// TwinCAT 3 PLC project PLC
// ProgramVersion: 3.1.4026.20
// CompilerDefines: VISU_USEPROPERTYINFO
// libraries:
//   Tc2_Standard, * (Beckhoff Automation GmbH)
//   Tc2_System, * (Beckhoff Automation GmbH)
//   Tc3_Vision, * (Beckhoff Automation GmbH)
//   VisuSymbols, 4.5.0.0 (System)
// project tree:
//   / GlobalTextList.TcGTLO, MAIN.TcPOU, PlcTask.TcTTO, Visualization Manager.TcVMO (not stored)
//   GVLs/ GVL.TcGVL
//   Source/debug/ CheckBounds.TcPOU (not stored)
//   Source/EL2574/DUT/ ST_EL2574_ExtendedMode.TcDUT, ST_EL2574_In.TcDUT, ST_EL2574_Out.TcDUT
//   Source/EL2574/ EL2574_ExtendedMode.TcPOU, I_EL2574_CommandMode.TcIO
//   Source/ImageSerializer/Base/ ImageSerializer.TcPOU
//   Source/ImageSerializer/Interfaces/ I_ImageSerializer.TcIO
//   Source/ImageSerializer/Matrix/ MatrixImageSerializer.TcPOU
//   Source/ImageSerializer/Null/ NullImageSerializer.TcPOU
//   Source/Library/Animation/ I_Animation.TcIO, SpriteSheetAnimationFrames.TcPOU
//   Source/Library/BlendModes/ BaseBlender.TcPOU, I_ImageBlender.TcIO, LerpMixer.TcPOU, MultiplyMixer.TcPOU
//   Source/Library/ Modulate.TcPOU
//   Source/Library/Scene/ Scene.TcPOU
//   Source/PixelReader/ EL2574PixelReader.TcPOU, I_PixelReader.TcIO
//   Source/ ST_Colors.TcDUT, U_Pixel.TcDUT
//   Source/Unwrappers/ I_Unwrapper.TcIO, RepeatUnwrap.TcPOU, ExtendUnwrap.TcPOU, ReflectUnwrap.TcPOU
//   VISUs/ UC_Slider.TcVIS, Visualization.TcVIS
// real-time tasks:
//   TASK PlcTask: cycle T#1ms, priority 20, ADS port 350
// I/O:
//   DEVICE Device 2 (EtherCAT), AmsNetId 192.168.1.242.3.1
//     Term 1 (EK1200) [EK1200-5000 EtherCAT Power supply (2A E-Bus)]
//       Term 3 (EL2574) [EL2574 4 Ch. Pixel LED Controller]
//         modules: SlotGroup 1 (Slot 1, 2) (1xASYNC), SlotGroup 1 (Slot 1, 2) (1xASYNC), SlotGroup 2 (Slot 3, 4) (EMPTY2), SlotGroup 2 (Slot 3, 4) (EMPTY2)
//       Term 3 (EL9011) [EL9011 End Terminal]
// variable links:
//   (this object) <-> Device 2 (EtherCAT)/Term 1 (EK1200)/Term 3 (EL2574)
//     PlcTask Inputs/MAIN.el2574_ch1.pdo.In/Busy <-> SlotGroup 1 (Slot 1, 2) (1xASYNC)/Status Channel 1/Status/Busy
//     PlcTask Inputs/MAIN.el2574_ch1.pdo.In/CommandAck <-> SlotGroup 1 (Slot 1, 2) (1xASYNC)/Status Channel 1/Status/Command Acknowledge
//     PlcTask Inputs/MAIN.el2574_ch1.pdo.In/CommandReject <-> SlotGroup 1 (Slot 1, 2) (1xASYNC)/Status Channel 1/Status/Command Reject
//     PlcTask Inputs/MAIN.el2574_ch1.pdo.In/Error <-> SlotGroup 1 (Slot 1, 2) (1xASYNC)/Status Channel 1/Status/Error
//     PlcTask Inputs/MAIN.el2574_ch1.pdo.In/InputCycleCounter <-> SlotGroup 1 (Slot 1, 2) (1xASYNC)/Status Channel 1/Status/Input Cycle Counter
//     PlcTask Inputs/MAIN.el2574_ch1.pdo.In/SendAck <-> SlotGroup 1 (Slot 1, 2) (1xASYNC)/Status Channel 1/Status/Send Acknowledge
//     PlcTask Inputs/MAIN.el2574_ch1.pdo.In/Transmit <-> SlotGroup 1 (Slot 1, 2) (1xASYNC)/Status Channel 1/Status/Transmit
//     PlcTask Inputs/MAIN.el2574_ch1.pdo.In/UpdateAck <-> SlotGroup 1 (Slot 1, 2) (1xASYNC)/Status Channel 1/Status/Update Acknowledge
//     PlcTask Inputs/MAIN.el2574_ch1.pdo.In/Warning <-> SlotGroup 1 (Slot 1, 2) (1xASYNC)/Status Channel 1/Status/Warning
//     PlcTask Outputs/MAIN.el2574_ch1.pdo.Out/Execute <-> SlotGroup 1 (Slot 1, 2) (1xASYNC)/Extended Channel 1/Extended Control/Execute
//     PlcTask Outputs/MAIN.el2574_ch1.pdo.Out/Index <-> SlotGroup 1 (Slot 1, 2) (1xASYNC)/Extended Channel 1/Extended Control/Index
//     PlcTask Outputs/MAIN.el2574_ch1.pdo.Out/Segment <-> SlotGroup 1 (Slot 1, 2) (1xASYNC)/Extended Channel 1/Extended Control/Segment
//     PlcTask Outputs/MAIN.el2574_ch1.pdo.Out/Send <-> SlotGroup 1 (Slot 1, 2) (1xASYNC)/Extended Channel 1/Extended Control/Send
//     PlcTask Outputs/MAIN.el2574_ch1.pdo.Out/Update <-> SlotGroup 1 (Slot 1, 2) (1xASYNC)/Extended Channel 1/Extended Control/Update
//     PlcTask Outputs/MAIN.el2574_ch1.pdo.Out/Write <-> SlotGroup 1 (Slot 1, 2) (1xASYNC)/Extended Channel 1/Extended Control/Write

CONFIGURATION PLC
    RESOURCE PLC ON TwinCAT3
        TASK PlcTask(INTERVAL := T#1ms, PRIORITY := 20);
        PROGRAM MAIN WITH PlcTask : MAIN;
    END_RESOURCE
END_CONFIGURATION

// ---- Source/EL2574/DUT/ST_EL2574_ExtendedMode.TcDUT
TYPE ST_EL2574_ExtendedMode :
	STRUCT
		In	AT %I* : ST_EL2574_In;
		Out AT %Q* : ST_EL2574_Out;
	END_STRUCT
END_TYPE

// ---- Source/EL2574/DUT/ST_EL2574_In.TcDUT
TYPE ST_EL2574_In :
	STRUCT
		Busy			  : BIT;
		Transmit		  : BIT;
		SendAck			  : BIT;
		UpdateAck		  : BIT;
		CommandAck		  : BIT;
		CommandReject	  : BIT;
		Warning			  : BIT;
		Error			  : BIT;
		InputCycleCounter : BYTE;
	END_STRUCT
END_TYPE

// ---- Source/EL2574/DUT/ST_EL2574_Out.TcDUT
TYPE ST_EL2574_Out :
	STRUCT
		Execute : BIT;
		Send	: BIT;
		Update	: BIT;
		Write	: BIT;
		Index	: USINT;
		Segment : ARRAY[0..7] OF UDINT;
	END_STRUCT
END_TYPE

// ---- Source/ST_Colors.TcDUT
TYPE ST_Colors :
	STRUCT
		Red	  : BYTE;
		Green : BYTE;
		Blue  : BYTE;
		White : BYTE;
	END_STRUCT
END_TYPE

// ---- Source/U_Pixel.TcDUT
TYPE U_Pixel : UNION
		Pdo	   : UDINT;
		Colors : ST_Colors;
	END_UNION
END_TYPE

// ---- GVLs/GVL.TcGVL
VAR_GLOBAL CONSTANT
	STRIP_LENGTH : UDINT := 12;
END_VAR

// ---- Source/EL2574/I_EL2574_CommandMode.TcIO
INTERFACE I_EL2574_CommandMode

METHOD PUBLIC ClearAll : I_EL2574_CommandMode
VAR_INPUT
END_VAR
END_METHOD

METHOD PUBLIC ColorGradient2Point : I_EL2574_CommandMode
VAR_INPUT
	StartPosition : UINT;
	NumberOfPixels : UINT;
	Color1 : STRING(9);
	Color2 : STRING(9);
END_VAR
END_METHOD

METHOD PUBLIC ColorGradient3Point : I_EL2574_CommandMode
VAR_INPUT
	StartPosition : UINT;
	NumberOfPixels : UINT;
	Color1 : STRING(9);
	Color2 : STRING(9);
	Color3 : STRING(9);
END_VAR
END_METHOD

METHOD PUBLIC ColorGradient4Point : I_EL2574_CommandMode
VAR_INPUT
	StartPosition : UINT;
	NumberOfPixels : UINT;
	Color1 : STRING(9);
	Color2 : STRING(9);
	Color3 : STRING(9);
	Color4 : STRING(9);
END_VAR
END_METHOD

METHOD PUBLIC CopyPixels : I_EL2574_CommandMode
VAR_INPUT
	StartPosition : UINT;
	NumberOfPixels : UINT;
	TargetPosition : UINT;
END_VAR
END_METHOD

METHOD PUBLIC FillColor : I_EL2574_CommandMode
VAR_INPUT
	StartPosition : UINT;
	NumberOfPixels : UINT;
	Red : USINT;
	Green : USINT;
	Blue : USINT;
	White : USINT;
END_VAR
END_METHOD

METHOD PUBLIC Invert : I_EL2574_CommandMode
VAR_INPUT
	StartPosition : UINT;
	NumberOfPixels : UINT;
END_VAR
END_METHOD

METHOD PUBLIC MovePixels : I_EL2574_CommandMode
VAR_INPUT
	StartPosition : UINT;
	NumberOfPixels : UINT;
	TargetPosition : UINT;
END_VAR
END_METHOD

METHOD PUBLIC RotateLeft : I_EL2574_CommandMode
VAR_INPUT
	StartPosition : UINT;
	NumberOfPixels : UINT;
	Shift : UINT;
END_VAR
END_METHOD

METHOD PUBLIC RotateRight : I_EL2574_CommandMode
VAR_INPUT
	StartPosition : UINT;
	NumberOfPixels : UINT;
	Shift : UINT;
END_VAR
END_METHOD

METHOD PUBLIC Send : I_EL2574_CommandMode
VAR_INPUT
END_VAR
END_METHOD

METHOD PUBLIC SendAndUpdate : I_EL2574_CommandMode
VAR_INPUT
END_VAR
END_METHOD

METHOD PUBLIC Update : I_EL2574_CommandMode
VAR_INPUT
END_VAR
END_METHOD

END_INTERFACE

// ---- Source/ImageSerializer/Interfaces/I_ImageSerializer.TcIO
INTERFACE I_ImageSerializer

METHOD PUBLIC ConnectTo
VAR_INPUT
	ImageSerializer : I_ImageSerializer;
END_VAR
END_METHOD

METHOD PUBLIC GetTotalSerializablePixelCount : UDINT
VAR_INPUT
END_VAR
END_METHOD

PROPERTY PUBLIC PixelCount : UDINT
GET
END_GET
END_PROPERTY

METHOD PUBLIC TryGetPixel : BOOL
VAR_INPUT
	PixelIndex : UDINT;
	Reader : I_PixelReader;
END_VAR
END_METHOD

METHOD PUBLIC UpdateImage
VAR_INPUT
	Source : ITcVnImage;
END_VAR
END_METHOD

END_INTERFACE

// ---- Source/Library/Animation/I_Animation.TcIO
INTERFACE I_Animation

PROPERTY PUBLIC CurrentFrameImage : ITcVnImage
GET
END_GET
END_PROPERTY

PROPERTY PUBLIC CurrentFrameIndex : UDINT
GET
END_GET
END_PROPERTY

PROPERTY PUBLIC IsAtLastFrame : BOOL
GET
END_GET
END_PROPERTY

METHOD PUBLIC MoveToStart
VAR_INPUT
END_VAR
END_METHOD

PROPERTY PUBLIC TotalFrameCount : UDINT
GET
END_GET
END_PROPERTY

METHOD PUBLIC TryMoveNext : BOOL
VAR_INPUT
END_VAR
END_METHOD

METHOD PUBLIC TryMovePrevious : BOOL
VAR_INPUT
END_VAR
END_METHOD

END_INTERFACE

// ---- Source/Library/BlendModes/I_ImageBlender.TcIO
INTERFACE I_ImageBlender

METHOD Mix
VAR_INPUT
	ImageBottomLayer : ITcVnImage;
	ImageTopLayer	 : ITcVnImage;
END_VAR
END_METHOD

END_INTERFACE

// ---- Source/PixelReader/I_PixelReader.TcIO
INTERFACE I_PixelReader

PROPERTY PUBLIC Value : Reference to TcVnVector4_LREAL
GET
END_GET
END_PROPERTY

END_INTERFACE

// ---- Source/Unwrappers/I_Unwrapper.TcIO
INTERFACE I_Unwrapper

METHOD Sample : BOOL
VAR_INPUT
	ImageWidth, ImageHeight	  : UDINT;
	XOffset, YOffset		  : UDINT;
END_VAR
END_METHOD

PROPERTY X : UDINT
GET
END_GET
END_PROPERTY

PROPERTY Y : UDINT
GET
END_GET
END_PROPERTY

END_INTERFACE

// ---- MAIN.TcPOU
PROGRAM MAIN
VAR
	// --- Sprite source images ---
	Black	   : SpriteSheetAnimationFrames(SpriteSheetFilePath := 'C:\temp\images\black_64x1.png', SpriteWidth := 64, SpriteHeight := 1, TotalSprites := 1, Columns := 1, Rows := 1);
	Red		   : SpriteSheetAnimationFrames(SpriteSheetFilePath := 'C:\temp\images\red_64x1.png', SpriteWidth := 64, SpriteHeight := 1, TotalSprites := 1, Columns := 1, Rows := 1);
	Blue	   : SpriteSheetAnimationFrames(SpriteSheetFilePath := 'C:\temp\images\blue_64x1.png', SpriteWidth := 64, SpriteHeight := 1, TotalSprites := 1, Columns := 1, Rows := 1);
	Green	   : SpriteSheetAnimationFrames(SpriteSheetFilePath := 'C:\temp\images\green_64x1.png', SpriteWidth := 64, SpriteHeight := 1, TotalSprites := 1, Columns := 1, Rows := 1);
	Background : SpriteSheetAnimationFrames(SpriteSheetFilePath := 'C:\temp\images\rainbow_gradient.png', SpriteWidth := 1000, SpriteHeight := 1, TotalSprites := 1, Columns := 1, Rows := 1);
	white	   : SpriteSheetAnimationFrames(SpriteSheetFilePath := 'C:\temp\images\whitealpha3_32_32.png', SpriteWidth := 32, SpriteHeight := 1, TotalSprites := 1, Columns := 1, Rows := 1);
	shortred   : SpriteSheetAnimationFrames(SpriteSheetFilePath := 'C:\temp\images\shortred_32_32.png', SpriteWidth := 32, SpriteHeight := 1, TotalSprites := 1, Columns := 1, Rows := 1);

	// --- Modulators (scroll/unwrap each source into a strip-length output) ---
	ModulateBackground : Modulate(Width := GVL.STRIP_LENGTH);
	ShortredModulator  : Modulate(Width := GVL.STRIP_LENGTH);
	WhiteModulator	   : Modulate(Width := GVL.STRIP_LENGTH);
	backgroundOffset   : UDINT;
	shortredOffset	   : UDINT;
	shortedRollOver	   : UDINT;
	whiteOffset		   : UDINT;
	whiteRollOver	   : UDINT;
	redOffset		   : UDINT;
	blueOffset		   : UDINT;
	greenOffset		   : UDINT;
	UpdateBackground   : BOOL;
	UpdateShortred	   : BOOL;
	UpdateWhite		   : BOOL;
	UpdateRed		   : BOOL;
	UpdateBlue		   : BOOL;
	UpdateGreen		   : BOOL;

	// --- Scene compositor ---
	MyScene : Scene;
	lerp	: LerpMixer;
	weight	: LREAL := 0.85;

	// --- Displayable image handles (for scope/HMI monitoring) ---
	SceneImage		  : ITcVnDisplayableImage;
	displayBackground : ITcVnDisplayableImage;
	displayShortred	  : ITcVnDisplayableImage;
	displayWhite	  : ITcVnDisplayableImage;
	displayRed		  : ITcVnDisplayableImage;
	displayBlue		  : ITcVnDisplayableImage;
	displayGreen	  : ITcVnDisplayableImage;

	// --- Animation timing ---
	Animate			 : BOOL := TRUE;
	AddBlackLayer	 : BOOL := FALSE;
	AnimateBackgroud : BOOL := TRUE;
	AddBackground	 : BOOL := TRUE;
	BackgroundRate	 : TON	:= (PT := T#80MS);
	AddShortedLayer	 : BOOL := TRUE;
	ShortredRate	 : TON	:= (PT := T#200MS);
	AddWhiteLayer	 : BOOL := TRUE;
	WhiteRate		 : TON	:= (PT := T#150MS);
	AddRedLayer		 : BOOL := FALSE;
	AddBlueLayer	 : BOOL := FALSE;
	AddGreenLayer	 : BOOL := FALSE;

	// --- Unwrap modes ---
	unwraptype			: UDINT;
	reflect				: ReflectUnwrap;
	RepeatNormal		: RepeatUnwrap;
	Extend				: ExtendUnwrap;
	width, height, x, y : UDINT; // reflect.Sample inputs

	// --- Hardware ---
	LEDStrip   : MatrixImageSerializer(Height := 1, Width := GVL.STRIP_LENGTH, X := 0, Y := 0, FlipX := FALSE, FlipY := FALSE, Rotate := FALSE);
	el2574_ch1 : EL2574_ExtendedMode(TotalPixels := GVL.STRIP_LENGTH);

	// --- Misc ---
	val	   : HRESULT;
	format : TcVnPixelFormat;
END_VAR

_AppInfo.KeepOutputsOnBP := TRUE;
// 1. LOAD GUARD — wait until all sprite sheets are ready
IF NOT Black.TryLoad() OR NOT Background.TryLoad() OR NOT shortred.TryLoad() OR NOT white.TryLoad() OR NOT Red.TryLoad() OR NOT Blue.TryLoad() OR NOT Green.TryLoad() THEN
	RETURN;
END_IF

// 2. ANIMATION TICK — advance offsets at each layer's own rate
ShortredRate(IN := NOT ShortredRate.Q AND Animate);
IF ShortredRate.Q THEN
	shortredOffset := shortredOffset + 1;
	IF shortredOffset >= shortedRollOver THEN
		shortredOffset := 0;
	END_IF

	UpdateShortred := TRUE;
END_IF

WhiteRate(IN := NOT WhiteRate.Q AND Animate);
IF WhiteRate.Q THEN
	whiteOffset := whiteOffset + 1;
	IF whiteOffset >= whiteRollOver THEN
		whiteOffset := 0;
	END_IF

	UpdateWhite := TRUE;
END_IF

BackgroundRate(IN := NOT BackgroundRate.Q AND Animate AND AnimateBackgroud);
IF BackgroundRate.Q THEN
	backgroundOffset := backgroundOffset + 1;
	UpdateBackground := TRUE;
END_IF

// 3. UNWRAP MODE SELECT — override shortred/white unwrapper at runtime
ModulateBackground.Unwrapper := reflect;
CASE unwraptype OF
	0:
		shortedRollOver				:= 32;
		whiteRollOver				:= 32;
		ShortredModulator.Unwrapper := RepeatNormal;
		WhiteModulator.Unwrapper	:= RepeatNormal;

	1:
		shortedRollOver				:= GVL.STRIP_LENGTH;
		whiteRollOver				:= GVL.STRIP_LENGTH;
		ShortredModulator.Unwrapper := reflect;
		WhiteModulator.Unwrapper	:= reflect;

	2:
		ShortredModulator.Unwrapper := Extend;
		WhiteModulator.Unwrapper	:= Extend;

END_CASE

// 4. MODULATE — scroll each source into a strip-length output frame
IF UpdateBackground OR NOT AnimateBackgroud THEN
	ModulateBackground.GetImage(Source		 := Background.CurrentFrameImage,
								SourceWidth	 := 1000,
								SourceHeight := 1,
								OutputWidth	 := GVL.STRIP_LENGTH,
								OutputHeight := 1,
								OffsetX		 := backgroundOffset,
								OffsetY		 := 0);

	UpdateBackground := FALSE;
END_IF

IF UpdateShortred THEN
	ShortredModulator.GetImage(shortred.CurrentFrameImage,
							   32,
							   1,
							   GVL.STRIP_LENGTH,
							   1,
							   shortredOffset,
							   0);

	UpdateShortred := FALSE;
END_IF

IF UpdateWhite THEN
	WhiteModulator.GetImage(white.CurrentFrameImage,
							32,
							1,
							GVL.STRIP_LENGTH,
							1,
							whiteOffset,
							0);

	UpdateWhite := FALSE;
END_IF

// 5. COMPOSE SCENE — stack layers onto background with lerp blend
IF NOT el2574_ch1.IsBusy THEN
	IF AddBlackLayer THEN
		MyScene.Initalize(Black.CurrentFrameImage);
	END_IF

	IF AddBackground THEN
		MyScene.Initalize(ModulateBackground.CurrentFrameImage);
	END_IF

	lerp.Weight := weight;
	
	IF AddWhiteLayer THEN
		MyScene.AddLayer(WhiteModulator.CurrentFrameImage, lerp);
	END_IF
	
	IF AddShortedLayer THEN
		MyScene.AddLayer(ShortredModulator.CurrentFrameImage, lerp);
	END_IF

	IF AddRedLayer THEN
		MyScene.AddLayer(Red.CurrentFrameImage, lerp);
	END_IF

	IF AddBlueLayer THEN
		MyScene.AddLayer(Blue.CurrentFrameImage, lerp);
	END_IF

	IF AddGreenLayer THEN
		MyScene.AddLayer(Green.CurrentFrameImage, lerp);
	END_IF

	LEDStrip.UpdateImage(MyScene.Image);
	el2574_ch1.TrySendPixelsFromSerializer(LEDStrip);

	// 6. COPY TO DISPLAY — push images to HMI/scope handles
	val := F_VN_CopyIntoDisplayableImage(MyScene.Image, SceneImage, s_ok);
	val := F_VN_CopyIntoDisplayableImage(ModulateBackground.CurrentFrameImage, displayBackground, s_ok);
	val := F_VN_CopyIntoDisplayableImage(ShortredModulator.CurrentFrameImage, displayShortred, s_ok);
	val := F_VN_CopyIntoDisplayableImage(WhiteModulator.CurrentFrameImage, displayWhite, s_ok);
END_IF

el2574_ch1.CyclicCall();

END_PROGRAM

// ---- Source/Library/Animation/SpriteSheetAnimationFrames.TcPOU
FUNCTION_BLOCK SpriteSheetAnimationFrames IMPLEMENTS I_Animation
VAR
	spriteSheetFilePath : T_MAXSTRING;
	spriteWidth			: UDINT;
	spriteHeight		: UDINT;
	totalSprites		: UDINT;
	columns				: UDINT;
	rows				: UDINT;
	spriteSheetImage	: ITcVnImage;
	readImage			: FB_VN_ReadImage;

	// animation variables
	_currentFrameIndex	 : UDINT;
	_currentFrameImage	 : ITcVnImage;
	_LoadedImageFromDisk : ITcVnDisplayableImage;
END_VAR

PROPERTY PUBLIC CurrentFrameImage : ITcVnImage
GET
CurrentFrameImage := _currentFrameImage;
END_GET
END_PROPERTY

PROPERTY PUBLIC CurrentFrameIndex : UDINT
GET
CurrentFrameIndex := _currentFrameIndex;
END_GET
END_PROPERTY

METHOD FB_init : BOOL
VAR_INPUT
	bInitRetains		: BOOL; // if TRUE, the retain variables are initialized (warm start / cold start)
	bInCopyCode			: BOOL; // if TRUE, the instance afterwards gets moved into the copy code (online change)
	SpriteSheetFilePath : T_MAXSTRING;
	SpriteWidth			: UDINT;
	SpriteHeight		: UDINT;
	TotalSprites		: UDINT;
	Columns				: UDINT;
	Rows				: UDINT;
END_VAR
THIS^.spriteSheetFilePath := SpriteSheetFilePath;
THIS^.spriteWidth		  := SpriteWidth;
THIS^.spriteHeight		  := SpriteHeight;
THIS^.totalSprites		  := TotalSprites;
THIS^.columns			  := Columns;
THIS^.rows				  := Rows;
END_METHOD

PROPERTY PUBLIC IsAtLastFrame : BOOL
GET
IF TotalFrameCount = 0 THEN
	IsAtLastFrame := TRUE;
	RETURN;
END_IF

IsAtLastFrame := CurrentFrameIndex = TotalFrameCount - 1;
END_GET
END_PROPERTY

METHOD PUBLIC MoveToStart
VAR_INPUT
END_VAR
_currentFrameIndex := 0;
TryGetSprite(_currentFrameIndex, _currentFrameImage);
END_METHOD

PROPERTY PUBLIC TotalFrameCount : UDINT
GET
TotalFrameCount := totalSprites;
END_GET
END_PROPERTY

METHOD PRIVATE TryGetSprite : BOOL
VAR_INPUT
	Index : UDINT;
	Destination : REFERENCE TO ITcVnImage;
END_VAR
VAR
	spriteX : UDINT;
	spriteY : UDINT;
	spriteColumn : UDINT;
	spriteRow : UDINT;
	result : HRESULT;
END_VAR
IF Index > TotalFrameCount - 1 THEN
	RETURN;
END_IF

spriteColumn := Index MOD columns;
spriteRow := Index / columns;

spriteX := spriteColumn * spriteWidth;
spriteY := spriteRow * spriteHeight;

result := F_VN_CopyImage(spriteSheetImage, _currentFrameImage, s_OK);
result := F_VN_SetRoi(spriteX, spriteY, spriteWidth, spriteHeight, _currentFrameImage, result);

TryGetSprite := Succeeded(result);
END_METHOD

METHOD PUBLIC TryLoad : BOOL
VAR
	i : UDINT;
END_VAR
// if we already have an image loaded, then we can early jump out as we know everything is done. 
IF spriteSheetImage <> 0 THEN
	TryLoad := TRUE;
	RETURN;
END_IF

IF spriteSheetFilePath = '' OR  spriteWidth = 0 OR spriteHeight = 0 OR totalSprites = 0 OR columns = 0 OR rows = 0 THEN
	// this is our sanity check, we return out if anything is bad.
	// if we pass this point we know we can use the variables confidently.
	RETURN;
END_IF

// we keep polling the read until an image is read.  If it faults due to error then we just sit here and never return true.
readImage(sFilePath := spriteSheetFilePath, ipDestImage := spriteSheetImage, bRead := TRUE, nTimeout := T#500MS);
IF readImage.bBusy THEN 
	RETURN;
END_IF

IF readImage.bError THEN 
	RETURN;
END_IF 

// at this point we should have an image, so we will do one final check before moving on.  
IF spriteSheetImage = 0 THEN
	RETURN;
END_IF

F_VN_CopyIntoDisplayableImage(ipSrcImage:=spriteSheetImage,ipDestImage:=_LoadedImageFromDisk,hrPrev:=S_OK);

// we have made it this far, which means we need to set the CurrentFrameImage to the first part of the image and report as done. 
MoveToStart();
TryLoad := TRUE;
END_METHOD

METHOD PUBLIC TryMoveNext : BOOL
VAR_INPUT
END_VAR
IF _currentFrameIndex = TotalFrameCount - 1 THEN
	RETURN;
END_IF

_currentFrameIndex := _currentFrameIndex + 1;
TryMoveNext := TryGetSprite(_currentFrameIndex, _currentFrameImage);
END_METHOD

METHOD PUBLIC TryMovePrevious : BOOL
VAR_INPUT
END_VAR
IF _currentFrameIndex = 0 THEN
	RETURN;
END_IF

_currentFrameIndex := _currentFrameIndex - 1;
TryMovePrevious := TryGetSprite(_currentFrameIndex, _currentFrameImage);
END_METHOD

END_FUNCTION_BLOCK

// ---- Source/Library/Modulate.TcPOU
FUNCTION_BLOCK Modulate
VAR
	_CurrentImage : ITcVnImage;
	_unwrapper	  : I_Unwrapper;
	value		  : HRESULT;
END_VAR

PROPERTY PUBLIC CurrentFrameImage : ITcVnImage
GET
CurrentFrameImage := _CurrentImage;
END_GET
END_PROPERTY

//FB_Init is always available implicitly and it is used primarily for initialization.
//The return value is not evaluated. For a specific influence, you can also declare the
//methods explicitly and provide additional code there with the standard initialization
//code. You can evaluate the return value.
METHOD FB_Init: BOOL
VAR_INPUT
    bInitRetains: BOOL; // TRUE: the retain variables are initialized (reset warm / reset cold)
    bInCopyCode: BOOL;  // TRUE: the instance will be copied to the copy code afterward (online change)
    Width: UDINT;       // Output image buffer width — pass GVL.STRIP_LENGTH
END_VAR
F_VN_CreateImage(_CurrentImage,
				 Width,
				 1,
				 ETcVnElementType.TCVN_ET_USINT,
				 4,
				 S_OK);
END_METHOD

METHOD GetImage
VAR_INPUT
	Source					  : ITcVnImage;
	SourceWidth, SourceHeight : UDINT;
	OutputWidth, OutputHeight : UDINT;
	OffsetX, Offsety		  : UDINT;
END_VAR

VAR
	x, y			   : UDINT;
	_SampleX, _SampleY : UDINT;
	currentPixel	   : TcVnVector4_LREAL;
END_VAR
FOR y := 0 TO OutputHeight - 1 DO
	FOR x := 0 TO OutputWidth - 1 DO
		_unwrapper.Sample(ImageWidth  := SourceWidth,
						  ImageHeight := SourceHeight,
						  XOffset	  := x + OffsetX,
						  YOffset	  := y + OffsetY);

		IF SUCCEEDED(F_VN_GetPixel(ipSrcImage := Source,
								   aValue	  := currentPixel,
								   nX		  := _unwrapper.X,
								   nY		  := _unwrapper.Y,
								   hrPrev	  := s_OK)) THEN
			value := F_VN_SetPixel(ipSrcImage := _CurrentImage,
						  aValue	 := currentPixel,
						  nX		 := x,
						  nY		 := y,
						  hrPrev	 := s_OK);
		END_IF
	END_FOR
END_FOR
END_METHOD

PROPERTY Unwrapper : I_Unwrapper
GET
Unwrapper := _unwrapper;
END_GET
SET
_unwrapper := Unwrapper;
END_SET
END_PROPERTY

END_FUNCTION_BLOCK

// ---- Source/Library/Scene/Scene.TcPOU
FUNCTION_BLOCK Scene
VAR
	sceneImage : ITcVnImage;
END_VAR

METHOD PUBLIC AddLayer
VAR_INPUT
	Source	  : ITcVnImage;
	BlendMode : I_ImageBlender;
END_VAR

VAR
	sourceHeight, currentHeight : UDINT;
	sourceWidth, currentWidth	: UDINT;
	x, y						: UDINT;
	currentPixel				: TcVnVector4_LREAL;
END_VAR
IF sceneImage = 0 THEN
	RETURN;
END_IF

IF Source = 0 THEN
	RETURN;
END_IF

IF FAILED(Source.GetHeight(sourceHeight)) THEN
	RETURN;
END_IF;

IF FAILED(sceneImage.GetHeight(currentHeight)) THEN
	RETURN;
END_IF;

IF FAILED(Source.GetWidth(sourceWidth)) THEN
	RETURN;
END_IF;

IF FAILED(sceneImage.GetWidth(currentWidth)) THEN
	RETURN;
END_IF;

IF sourceHeight > currentHeight THEN
	RETURN;
END_IF

IF sourceWidth > currentWidth THEN
	RETURN;
END_IF

IF BlendMode = 0 THEN
	RETURN;
END_IF

BlendMode.Mix(ImageBottomLayer := sceneImage, ImageTopLayer := Source);
END_METHOD

PROPERTY PUBLIC Image : ITcVnImage
GET
Image := sceneImage;
END_GET
END_PROPERTY

METHOD PUBLIC Initalize
VAR_INPUT
	Source : ITcVnImage;
END_VAR
F_VN_CopyImage(Source, sceneImage, s_OK);
END_METHOD

END_FUNCTION_BLOCK

// ---- Source/Library/BlendModes/LerpMixer.TcPOU
FUNCTION_BLOCK LerpMixer Extends BaseBlender
VAR
	_Weight : LREAL;
END_VAR

METHOD Mix
VAR_INPUT
	ImageBottomLayer : ITcVnImage;
	ImageTopLayer	 : ITcVnImage;
END_VAR
VAR_INST
	newWeight : LREAL;
END_VAR
VAR
	bottomPixel, topPixel, newPixel : TcVnVector4_LREAL;
	x, y							: UDINT;
	
	val								: HRESULT;
END_VAR
IF NOT InputCheck(ImageBottomLayer, ImageTopLayer) THEN
	RETURN;
END_IF

IF _Weight < 0 OR _Weight > 1 THEN
	RETURN;
END_IF

FOR x := 0 TO ImageOneWidth - 1 DO
	FOR y := 0 TO ImageOneHeight - 1 DO
		F_VN_GetPixel(ipSrcImage := ImageBottomLayer,
					  aValue	 := bottomPixel,
					  nX		 := x,
					  nY		 := y,
					  hrPrev	 := s_OK);

		F_VN_GetPixel(ipSrcImage := ImageTopLayer,
					  aValue	 := topPixel,
					  nX		 := x,
					  nY		 := y,
					  hrPrev	 := s_OK);
		//newWeight := topPixel[3] / 255.0;
		 newWeight := (_Weight) * (topPixel[3] / 255.0);
		 
		newPixel[0] := (topPixel[0] * newWeight) + (bottomPixel[0] * (1.0 - newWeight));
		newPixel[1] := (topPixel[1] * newWeight) + (bottomPixel[1] * (1.0 - newWeight));
		newPixel[2] := (topPixel[2] * newWeight) + (bottomPixel[2] * (1.0 - newWeight));  
		//newPixel[0] := ABS(bottomPixel[0] - topPixel[0]) * (newWeight) + bottomPixel[0];
// 		newPixel[1] := ABS(bottomPixel[1] - topPixel[1]) * (newWeight) + bottomPixel[1];
// 		newPixel[2] := ABS(bottomPixel[2] - topPixel[2]) * (newWeight) + bottomPixel[2];
		newPixel[3] := 255;
		//newPixel[3] := (bottomPixel[3] - topPixel[3]) * (_Weight) + topPixel[3];
		val := F_VN_SetPixel(ipSrcImage := ImageBottomLayer,
					  aValue	 := newPixel,
					  nX		 := x,
					  nY		 := y,
					  hrPrev	 := s_OK);
	END_FOR
END_FOR
END_METHOD

// % interpolation between the two images
PROPERTY Weight : LREAL
GET
Weight := _Weight;
END_GET
SET
_Weight := Weight;
END_SET
END_PROPERTY

END_FUNCTION_BLOCK

// ---- Source/Library/BlendModes/BaseBlender.TcPOU
FUNCTION_BLOCK ABSTRACT BaseBlender IMPLEMENTS I_ImageBlender
VAR
	ImageOneHeight, ImageOneWidth : UDINT;
	ImageTwoHeight, ImageTwoWidth : UDINT;
END_VAR

METHOD PROTECTED InputCheck : BOOL
VAR_INPUT	
	ImageOne	: ITcVnImage;
	ImageTwo	: ITcVnImage;
END_VAR
IF ImageOne = 0 OR ImageTwo = 0 THEN
	RETURN;
END_IF

IF FAILED(ImageOne.GetHeight(imageOneHeight)) THEN
	RETURN;
END_IF;

IF FAILED(ImageTwo.GetHeight(imageTwoHeight)) THEN
	RETURN;
END_IF;

IF FAILED(ImageOne.GetWidth(ImageOneWidth)) THEN
	RETURN;
END_IF;

IF FAILED(ImageTwo.GetWidth(ImageTwoWidth)) THEN
	RETURN;
END_IF;

IF ImageOneHeight <> ImageTwoHeight THEN
	RETURN;
END_IF

IF ImageOneWidth <> ImageTwoWidth THEN
	RETURN;
END_IF

InputCheck := TRUE;
END_METHOD

METHOD ABSTRACT Mix
VAR_INPUT
	ImageBottomLayer : ITcVnImage;
	ImageTopLayer	 : ITcVnImage;
END_VAR
END_METHOD

END_FUNCTION_BLOCK

// ---- Source/Unwrappers/ReflectUnwrap.TcPOU
FUNCTION_BLOCK ReflectUnwrap IMPLEMENTS I_Unwrapper
VAR
	_x : UDINT;
	_y : UDINT;
END_VAR

METHOD Sample : BOOL
VAR_INPUT
	ImageWidth	: UDINT;
	ImageHeight : UDINT;
	XOffset		: UDINT;
	YOffset		: UDINT;
END_VAR

VAR_INST
	factor : UDINT;
	even   : DINT;
END_VAR
even := TRUNC((XOffset) / (ImageWidth)) MOD 2;
IF even = 0 THEN
	_x := XOffset MOD ImageWidth;
ELSIF even = 1 THEN
	_x := ImageWidth - 1 - (XOffset MOD ImageWidth);
END_IF

_y	   := YOffset MOD ImageHeight;
Sample := TRUE;
END_METHOD

PROPERTY X : UDINT
GET
X := _x;
END_GET
END_PROPERTY

PROPERTY Y : UDINT
GET
Y := _y;
END_GET
END_PROPERTY

END_FUNCTION_BLOCK

// ---- Source/Unwrappers/RepeatUnwrap.TcPOU
FUNCTION_BLOCK RepeatUnwrap IMPLEMENTS I_Unwrapper
VAR
	_x : UDINT;
	_y : UDINT;
END_VAR

METHOD Sample : BOOL
VAR_INPUT
	ImageWidth	: UDINT;
	ImageHeight	: UDINT;
	XOffset	: UDINT;
	YOffset	: UDINT;
END_VAR
_x	   := XOffset MOD ImageWidth;
_y	   := YOffset MOD ImageHeight;
Sample := TRUE;
END_METHOD

PROPERTY X : UDINT
GET
X := _x;
END_GET
END_PROPERTY

PROPERTY Y : UDINT
GET
Y := _y;
END_GET
END_PROPERTY

END_FUNCTION_BLOCK

// ---- Source/Unwrappers/ExtendUnwrap.TcPOU
FUNCTION_BLOCK ExtendUnwrap IMPLEMENTS I_Unwrapper
VAR
	_x : UDINT;
	_y : UDINT;
END_VAR

METHOD Sample : BOOL
VAR_INPUT
	ImageWidth	: UDINT;
	ImageHeight	: UDINT;
	XOffset	: UDINT;
	YOffset	: UDINT;
END_VAR
_x	   := MIN(ImageWidth - 1, XOffset);
_y	   := MIN(ImageHeight - 1, YOffset);
Sample := TRUE;
END_METHOD

PROPERTY X : UDINT
GET
X := _x;
END_GET
END_PROPERTY

PROPERTY Y : UDINT
GET
Y := _y;
END_GET
END_PROPERTY

END_FUNCTION_BLOCK

// ---- Source/ImageSerializer/Matrix/MatrixImageSerializer.TcPOU
FUNCTION_BLOCK MatrixImageSerializer EXTENDS ImageSerializer
VAR
	height		   : UDINT;
	width		   : UDINT;
	x			   : UDINT;
	y			   : UDINT;
	flipRequired   : BOOL;
	flipAxis	   : ETcVnFlipAxis;
	rotateRequired : BOOL;
	rotateAngle	   : ETcVnRotationAngle;
	image		   : ITcVnImage;
	live		   : ITcVnDisplayableImage; // used in this demo to show the image for the matrix
	_pixelCount	   : UDINT;
END_VAR

METHOD FB_init : BOOL
VAR_INPUT
	bInitRetains : BOOL; // if TRUE, the retain variables are initialized (warm start / cold start)
	bInCopyCode	 : BOOL; // if TRUE, the instance afterwards gets moved into the copy code (online change)
	Height		 : UDINT;
	Width		 : UDINT;
	X			 : UDINT;
	Y			 : UDINT;
	FlipX		 : BOOL;
	FlipY		 : BOOL;
	Rotate		 : BOOL;
END_VAR
THIS^.height := Height;
THIS^.width := Width;
THIS^.x := X;
THIS^.y := Y;

IF FlipX AND FlipY THEN
	flipAxis := ETcVnFlipAxis.TCVN_FA_XY;
	flipRequired := TRUE;
ELSIF FlipX THEN
	flipAxis := ETcVnFlipAxis.TCVN_FA_X;
	flipRequired := TRUE;
ELSIF FlipY THEN
	flipAxis := ETcVnFlipAxis.TCVN_FA_Y;
	flipRequired := TRUE;
END_IF

IF Rotate THEN
	rotateRequired := TRUE;
	rotateAngle := ETcVnRotationAngle.TCVN_RA_90_DEG;
END_IF

Initialize();
END_METHOD

METHOD PRIVATE Initialize
VAR_INPUT
END_VAR
_pixelCount := width * height;
END_METHOD

METHOD PROTECTED OnTryGetPixel : BOOL
VAR_INPUT
	PixelIndex : UDINT;
	Reader	   : I_PixelReader;
END_VAR

VAR
	xPosition : UDINT;
	yPosition : UDINT;
END_VAR
IF width = 0 OR height = 0 THEN
	RETURN;
END_IF

xPosition := PixelIndex MOD width;
yPosition := PixelIndex / width;

// If it's an odd row, reverse the direction
IF yPosition MOD 2 = 1 THEN 
    xPosition := (width - 1) - xPosition;
END_IF

OnTryGetPixel := succeeded(F_VN_GetPixel(image, Reader.Value, xPosition, yPosition, s_OK));
END_METHOD

METHOD PROTECTED OnUpdateImage
VAR_INPUT
	Source : ITcVnImage;
END_VAR
VAR
	result : HRESULT;
END_VAR
result := F_VN_CopyImage(Source, image, s_OK);
result := F_VN_SetRoi(x, y, width, height, image, result);

IF flipRequired THEN
	result := F_VN_FlipImage(image, image, flipAxis, result);	
END_IF

IF rotateRequired THEN
	result := F_VN_RotateImage(image, image, rotateAngle, result);	
END_IF

IF Succeeded(result) THEN
	F_VN_CopyIntoDisplayableImage(image, live, s_ok);
	RETURN;
END_IF

// there was an error, so best to clear the internal image as it's no longer valid.
// but only if there was an image there in fht first place.

IF image = 0 THEN
	RETURN;
END_IF

image.TcRelease();
image := 0;
END_METHOD

{attribute 'monitoring' := 'call'}
PROPERTY PUBLIC PixelCount : UDINT
GET
PixelCount := _pixelCount;
END_GET
END_PROPERTY

END_FUNCTION_BLOCK

// ---- Source/ImageSerializer/Base/ImageSerializer.TcPOU
FUNCTION_BLOCK ABSTRACT ImageSerializer IMPLEMENTS I_ImageSerializer
VAR
	// using the null object pattern so that you no longer need to check to see if next is <> 0
	nullImageSerializer : NullImageSerializer;
	next : I_ImageSerializer := nullImageSerializer;
END_VAR

METHOD PUBLIC ConnectTo
VAR_INPUT
	ImageSerializer : I_ImageSerializer;
END_VAR
IF ImageSerializer = 0  THEN
	next := nullImageSerializer;
END_IF

IF ImageSerializer = next THEN
	RETURN;
END_IF

next := ImageSerializer;
END_METHOD

METHOD PUBLIC GetTotalSerializablePixelCount : UDINT
VAR_INPUT
END_VAR
GetTotalSerializablePixelCount := PixelCount + NextSerializer.GetTotalSerializablePixelCount();
END_METHOD

PROPERTY PUBLIC NextSerializer : I_ImageSerializer
GET
NextSerializer := next;
END_GET
END_PROPERTY

METHOD PROTECTED ABSTRACT OnTryGetPixel : BOOL
VAR_INPUT
	PixelIndex : UDINT;
	Reader : I_PixelReader;
END_VAR
END_METHOD

METHOD PROTECTED ABSTRACT OnUpdateImage
VAR_INPUT
	Source : ITcVnImage;
END_VAR
END_METHOD

PROPERTY PUBLIC ABSTRACT PixelCount : UDINT
GET
END_GET
END_PROPERTY

METHOD PUBLIC TryGetPixel : BOOL
VAR_INPUT
	PixelIndex : UDINT;
	Reader : I_PixelReader;
END_VAR
VAR
	newPixelIndex : UDINT;
END_VAR
IF PixelIndex > PixelCount - 1 THEN
	newPixelIndex := PixelIndex - PixelCount;
	TryGetPixel := NextSerializer.TryGetPixel(newPixelIndex, Reader);
	RETURN;
END_IF

TryGetPixel := OnTryGetPixel(PixelIndex, Reader);
END_METHOD

METHOD PUBLIC UpdateImage
VAR_INPUT
	Source : ITcVnImage;
END_VAR
IF Source = 0 THEN
	RETURN;
END_IF

OnUpdateImage(Source);
NextSerializer.UpdateImage(Source);
END_METHOD

END_FUNCTION_BLOCK

// ---- Source/ImageSerializer/Null/NullImageSerializer.TcPOU
FUNCTION_BLOCK NullImageSerializer IMPLEMENTS I_ImageSerializer
VAR
END_VAR

METHOD PUBLIC ConnectTo
VAR_INPUT
	ImageSerializer : I_ImageSerializer;
END_VAR
END_METHOD

METHOD PUBLIC GetTotalSerializablePixelCount : UDINT
VAR_INPUT
END_VAR
GetTotalSerializablePixelCount := 0;
END_METHOD

PROPERTY PUBLIC PixelCount : UDINT
GET
PixelCount := 0;
END_GET
END_PROPERTY

METHOD PUBLIC TryGetPixel : BOOL
VAR_INPUT
	PixelIndex : UDINT;
	Reader : I_PixelReader;
END_VAR
TryGetPixel := FALSE;
END_METHOD

METHOD PUBLIC UpdateImage
VAR_INPUT
	Source : ITcVnImage;
END_VAR
END_METHOD

END_FUNCTION_BLOCK

// ---- Source/EL2574/EL2574_ExtendedMode.TcPOU
FUNCTION_BLOCK EL2574_ExtendedMode
VAR
	totalPixels		 : UDINT;
	pdo				 : ST_EL2574_ExtendedMode;
	sendBuffer		 : ARRAY[0..MAX_PIXELS - 1] OF U_Pixel;//UDINT;
	sendSegmentCount : USINT;
	currentSegment	 : USINT;
	state			 : (IDLE,
		INITIALIZING,
		SEND_SEGMENT,
		TRIGGER_FRAME_SEND,
		WAIT_FOR_FRAME_SEND_COMPLETE,
		ERROR);
END_VAR

VAR CONSTANT
	MAX_PIXELS : UDINT := 2048;
END_VAR

METHOD PRIVATE CreateSendBufferFromSerializer
VAR_INPUT
	ImageSerializer : I_ImageSerializer;
END_VAR
VAR
	currentPixel : UDINT := 0;
	pixelReader : EL2574PixelReader;
END_VAR
WHILE ImageSerializer.TryGetPixel(currentPixel, pixelReader) DO
	sendBuffer[currentPixel].Pdo := pixelReader.ReadAsUdint();
	currentPixel := currentPixel + 1;
END_WHILE
END_METHOD

METHOD PUBLIC CyclicCall
VAR_INPUT
END_VAR
VAR
	totalSegments : UDINT;
END_VAR
CASE state OF
	
	IDLE : RETURN;
	ERROR : RETURN;
	
	INITIALIZING :
	
		// initialize local variables
		currentSegment := 0;
		totalSegments := totalPixels / 8;
		sendSegmentCount := UDINT_TO_USINT(totalSegments);
	
		// reset the card to a known state		
		pdo.Out.Index := 0;
		pdo.Out.Send := FALSE;
		pdo.Out.Update := FALSE;
		pdo.Out.Write := FALSE;
		pdo.out.Segment[0] := 0;
		pdo.out.Segment[1]:= 0;
		pdo.out.Segment[2]:= 0;
		pdo.out.Segment[3]:= 0;
		pdo.out.Segment[4]:= 0;
		pdo.out.Segment[5]:= 0;
		pdo.out.Segment[6]:= 0;
		pdo.out.Segment[7]:= 0;
		
		// start sending....
		state := SEND_SEGMENT;

	SEND_SEGMENT :
		
		pdo.Out.Index := currentSegment;
		pdo.Out.Segment[0] := sendBuffer[currentSegment * 8 + 0].Pdo;
		pdo.Out.Segment[1] := sendBuffer[currentSegment * 8 + 1].Pdo;
		pdo.Out.Segment[2] := sendBuffer[currentSegment * 8 + 2].Pdo;
		pdo.Out.Segment[3] := sendBuffer[currentSegment * 8 + 3].Pdo;
		pdo.Out.Segment[4] := sendBuffer[currentSegment * 8 + 4].Pdo;
		pdo.Out.Segment[5] := sendBuffer[currentSegment * 8 + 5].Pdo;
		pdo.Out.Segment[6] := sendBuffer[currentSegment * 8 + 6].Pdo;
		pdo.Out.Segment[7] := sendBuffer[currentSegment * 8 + 7].Pdo;
		pdo.Out.Write := TRUE;
		pdo.Out.Execute := NOT pdo.Out.Execute;
				
		
		IF currentSegment = sendSegmentCount THEN
			state := TRIGGER_FRAME_SEND;
		ELSE
			currentSegment := currentSegment + 1;
		END_IF
		
	TRIGGER_FRAME_SEND : 
			
		pdo.Out.Write := FALSE;
		pdo.Out.Update := TRUE;
		pdo.Out.Send := TRUE;
		pdo.Out.Execute := NOT pdo.Out.Execute;	
		
		state := WAIT_FOR_FRAME_SEND_COMPLETE;
		
	WAIT_FOR_FRAME_SEND_COMPLETE:
	
		IF NOT pdo.In.Busy THEN
			pdo.out.Update := FALSE;
			pdo.out.Send := FALSE;
			state := IDLE;
		END_IF

		
END_CASE
END_METHOD

METHOD FB_init : BOOL
VAR_INPUT
	bInitRetains : BOOL; // if TRUE, the retain variables are initialized (warm start / cold start)
	bInCopyCode : BOOL;  // if TRUE, the instance afterwards gets moved into the copy code (online change)
	TotalPixels : UDINT;
END_VAR
This^.totalPixels := TotalPixels;
END_METHOD

PROPERTY PUBLIC HasError : BOOL
GET
HasError := state = Error;
END_GET
END_PROPERTY

PROPERTY PUBLIC IsBusy : BOOL
GET
IsBusy := not(state = IDLE or_else state = ERROR);
END_GET
END_PROPERTY

METHOD PRIVATE ResetSendBuffer
VAR_INPUT
END_VAR
memset(ADR(sendBuffer), 0,SIZEOF(sendBuffer));
END_METHOD

METHOD PUBLIC TrySendClearAll : BOOL
VAR_INPUT
END_VAR
IF IsBusy THEN 
	RETURN;
END_IF

state := INITIALIZING;

ResetSendBuffer();
TrySendClearAll := TRUE;
END_METHOD

METHOD PUBLIC TrySendPixelsFromSerializer : BOOL
VAR_INPUT
	ImageSerializer : I_ImageSerializer;
END_VAR
IF IsBusy THEN 
	RETURN;
END_IF

IF ImageSerializer.GetTotalSerializablePixelCount() > totalPixels THEN 
	RETURN;
END_IF

state := INITIALIZING;

ResetSendBuffer();
CreateSendBufferFromSerializer(ImageSerializer);
TrySendPixelsFromSerializer := TRUE;
END_METHOD

END_FUNCTION_BLOCK

// ---- Source/PixelReader/EL2574PixelReader.TcPOU
FUNCTION_BLOCK EL2574PixelReader IMPLEMENTS I_PixelReader
VAR
	pixelValue : TcVnVector4_LREAL;
END_VAR

METHOD PUBLIC ReadAsUdint : UDINT
VAR_INPUT
END_VAR

VAR
	pixel		: ARRAY[0..3] OF BYTE;
	pixelAsUint : UDINT;
END_VAR
pixel[0] := LREAL_TO_BYTE(value[0]);
pixel[1] := LREAL_TO_BYTE(value[1]);
pixel[2] := LREAL_TO_BYTE(value[2]);
//pixel[3] := LREAL_TO_BYTE(value[3]);
pixel[3]:=0;

memcpy(ADR(pixelAsUint), ADR(pixel),SIZEOF(pixelAsUint));
ReadAsUdint := pixelAsUint;
END_METHOD

PROPERTY PUBLIC Value : Reference to TcVnVector4_LREAL
GET
Value ref= pixelValue;
END_GET
END_PROPERTY

END_FUNCTION_BLOCK

// ---- Source/Library/BlendModes/MultiplyMixer.TcPOU
FUNCTION_BLOCK MultiplyMixer Extends BaseBlender
VAR
END_VAR

METHOD Mix
VAR_INPUT
	ImageBottomLayer : ITcVnImage;
	ImageTopLayer	 : ITcVnImage;
END_VAR
IF NOT InputCheck(ImageBottomLayer, ImageTopLayer) THEN
	RETURN;
END_IF

F_VN_MultiplyImages(ipSrcImage1 := ImageBottomLayer,
					ipSrcImage2 := ImageTopLayer,
					ipDestImage := ImageTopLayer,
					hrPrev		:= s_OK);
END_METHOD

END_FUNCTION_BLOCK

// ---- GlobalTextList.TcGTLO
TEXTLIST GlobalTextList
  561 = '%f'
  59 = '%s'
  337 = 'Animate'
  988 = 'Background'
  433 = 'Current'
  748 = 'Enable'
  273 = 'Lerp weight'
  201 = 'Start of window'
  393 = 'Voltage'
END_TEXTLIST

// ---- VISUs/UC_Slider.TcVIS
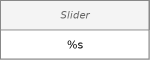
VISUALIZATION UC_Slider  // 150x60
VAR_IN_OUT
	PT		:TIME;
END_VAR
VAR_INPUT
	Start,End,MainScale	:UDINT;
	Label				:STRING;
END_VAR
    Slider (0,0 150x30), variable: PT, scale 0..1000
    Textfield (0,30 150x30), "%s", text variable: Label
END_VISUALIZATION

// ---- VISUs/Visualization.TcVIS
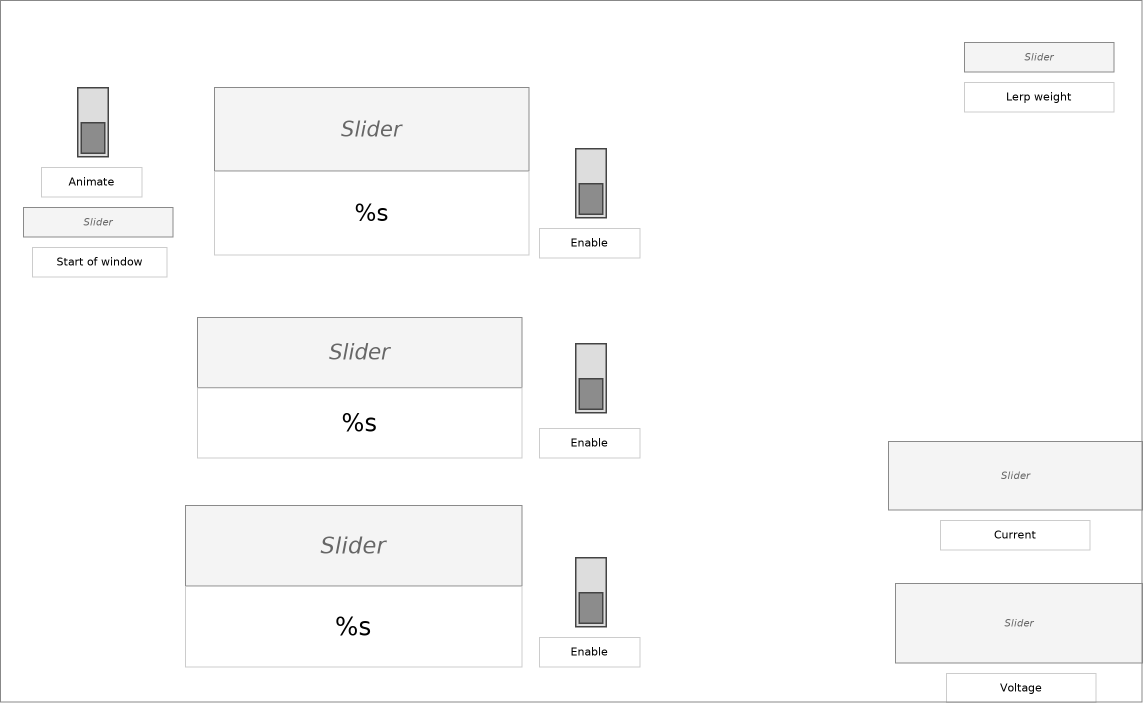
VISUALIZATION Visualization  // 1143x703
    Frame (214,87 315x168)
        shows UC_Slider(PT := MAIN.BackgroundRate.PT, Start := 1, End := 150, Label := 'Background')
    Frame (197,317 325x141)
        shows UC_Slider(PT := MAIN.WhiteRate.PT, Start := 1, End := 75, Label := 'White')
    Frame (185,505 337x162)
        shows UC_Slider(PT := MAIN.ShortredRate.PT, Start := 1, End := 75, Label := 'Shorted')
    DipSwitch (556,148 70x70), variable: MAIN.AddBackground, behaviour: TOGGLE, style: Switch-DipSwitch-Gray
    DipSwitch (556,557 70x70), variable: MAIN.AddShortedLayer, behaviour: TOGGLE, style: Switch-DipSwitch-Gray
    DipSwitch (556,343 70x70), variable: MAIN.AddWhiteLayer, behaviour: TOGGLE, style: Switch-DipSwitch-Gray
    DipSwitch (58,87 70x70), variable: MAIN.AnimateBackgroud, behaviour: TOGGLE, style: Switch-DipSwitch-Gray
    Slider (964,42 150x30), variable: MAIN.weight, scale 0..1
    Textfield (964,82 150x30), "Lerp weight"
    Textfield (41,167 101x30), "Animate"
    Slider (888,441 255x69), variable: MAIN.WhiteRate.PT, scale 1..75
    Slider (895,583 248x80), variable: MAIN.weight, scale 0..1
    Textfield (940,520 150x30), "Current"
    Textfield (946,673 150x30), "Voltage"
    Slider (23,207 150x30), variable: MAIN.backgroundOffset, scale 0..1000
    Textfield (539,228 101x30), "Enable"
    Textfield (539,428 101x30), "Enable"
    Textfield (539,637 101x30), "Enable"
    Textfield (32,247 135x30), "Start of window"
END_VISUALIZATION
